FUNCTION_BLOCK CL_DELAY (* Clocked delayed propagation of an event-Cancellable, Locally Clocked *)
  (* Standard: 61499-2; ApplicationDomain: Simulation; Function: Delay *)
  (* Version 0.0, 2004-09-23, JHC, Rockwell Automation *)
  (* Compiler header: package fb.rt.mva; import fb.rt.net.*; *)
  (* Compiler Java Sun JDK 1.4.2 *)
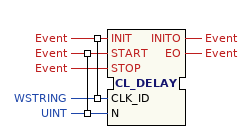
  EVENT_INPUT
    INIT WITH CLK_ID; (* Initialization Request *)
    START WITH N; (* Begin Delay *)
    STOP; (* Cancel Delay *)
  END_EVENT
  EVENT_OUTPUT
    INITO; (* Initialization Confirm *)
    EO; (* Delayed Event *)
  END_EVENT
  VAR_INPUT
    CLK_ID : WSTRING := "SIM_CLK"; (* Simulation Clock Channel ID *)
    N : UINT; (* Delay Time in Clock Cycles *)
  END_VAR
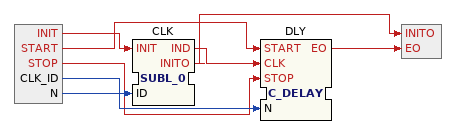
  FBS
    DLY : C_DELAY;
    CLK : SUBL_0;
  END_FBS
  EVENT_CONNECTIONS
    START TO DLY.START;
    DLY.EO TO EO;
    INIT TO CLK.INIT;
    CLK.IND TO DLY.CLK;
    STOP TO DLY.STOP;
    CLK.INITO TO INITO;
  END_CONNECTIONS
  DATA_CONNECTIONS
    N TO DLY.N;
    CLK_ID TO CLK.ID;
  END_CONNECTIONS
END_FUNCTION_BLOCK
